Staubli VAL3: cartStatus.pgx

public program cartStatus(num x_nCartConnFlag, num x_nLastMsgAge)
begin

  // update cartesian status on port 11001

  switch x_nCartConnFlag
    case -1
      userPageSet("uxMonitor", "lblCartState", "innerHTML", "connection lost")
    break
    case 0
      userPageSet("uxMonitor", "lblCartState", "innerHTML", "not connected")
    break
    case 1
      userPageSet("uxMonitor", "lblCartState", "innerHTML", "connected")
    break
    default
      userPageSet("uxMonitor", "lblCartState", "innerHTML", "not connected")
    break
  endSwitch

  if (x_nLastMsgAge < 0)
    userPageSet("uxMonitor", "lblCartAge", "innerHTML", "last msg: n/a")
  else
    userPageSet("uxMonitor", "lblCartAge", "innerHTML", "last msg: " + toString(".1", x_nLastMsgAge) + " s")
  endIf

end
